{attribute 'GeneratedUsingTerminal: KL1312'}
{attribute addProperty BoxType "KL1312"}
{attribute addProperty Description ""}
{attribute addProperty Physics ""}
{attribute addProperty Id "Channel_1AT %I*Channel_87C95E760Channel_2AT %I*Channel_87C95E760"}
{attribute addProperty CRC "3141065359"}
{attribute addProperty Size "0"}
TYPE KL1312_BB38DA8F :
STRUCT
	{attribute addProperty Name "Channel_1"}
	Channel_1 : Channel_87C95E76;
	{attribute addProperty Name "Channel_2"}
	Channel_2 : Channel_87C95E76;
END_STRUCT
END_TYPE

(* stored: Version 1.2.0.0, ProductVersion 3.1.4024.9
   DUT KL1312_BB38DA8F: Id {7da7e28a-9251-4bae-9ebb-458b9a877350} *)
